FUNCTION_BLOCK BUTTON (* Composite Function Block Type *)
  (* Standard: 61499-2 *)
  (* Version 0.0, 19/11/2012, vvya002, nxtControl GmbH, template *)
  PACKAGE Main;
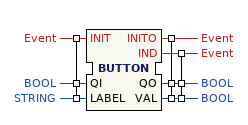
  EVENT_INPUT
    INIT WITH QI, LABEL; (* Initialization Request *)
  END_EVENT
  EVENT_OUTPUT
    INITO WITH QO, VAL; (* Initialization Confirm *)
    IND WITH QO, VAL; (* Execution Confirmation *)
  END_EVENT
  VAR_INPUT
    QI : BOOL; (* Input event qualifier *)
    LABEL : STRING;
  END_VAR
  VAR_OUTPUT
    QO : BOOL; (* Output event qualifier *)
    VAL : BOOL;
  END_VAR
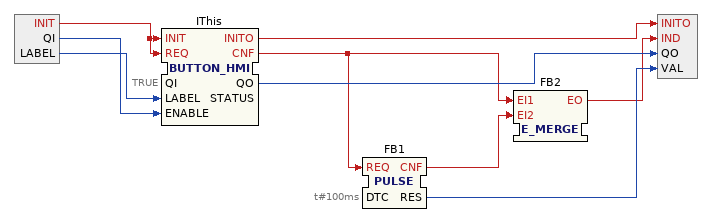
  FBS
    IThis : BUTTON_HMI(QI := TRUE);
    FB1 : PULSE(DTC := t#100ms);
    FB2 : E_MERGE;
  END_FBS
  EVENT_CONNECTIONS
    INIT TO IThis.INIT;
    INIT TO IThis.REQ;
    IThis.INITO TO INITO;
    IThis.CNF TO FB2.EI1;
    IThis.CNF TO FB1.REQ;
    FB1.CNF TO FB2.EI2;
    FB2.EO TO IND;
  END_CONNECTIONS
  DATA_CONNECTIONS
    LABEL TO IThis.LABEL;
    QI TO IThis.ENABLE;
    IThis.QO TO QO;
    FB1.RES TO VAL;
  END_CONNECTIONS
END_FUNCTION_BLOCK
